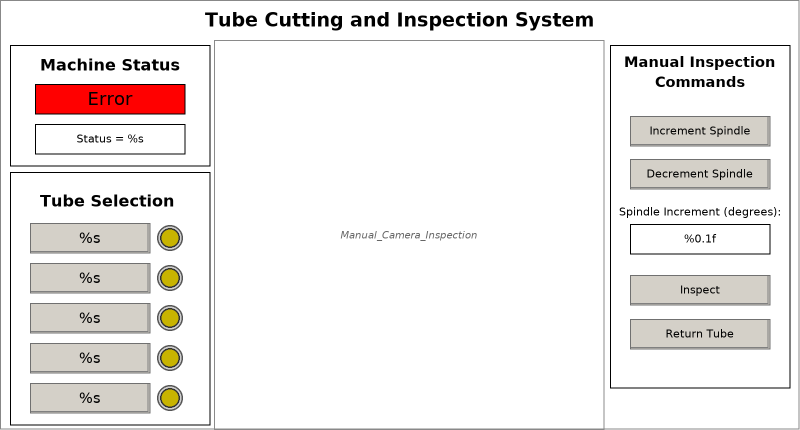
VISUALIZATION Manual_Inspect  // 800x430
    Rectangle (610,45 180x343)
    Frame (214,40 390x390)
        shows Manual_Camera_Inspection()
    Rectangle (10,172 200x253)
    Label (10,186 200x30), "Tube Selection"
    Button (30,223 120x30), "%s", text variable: MAIN.TubeSelection[1].ProductName
        OnMouseClick: execute {
            MAIN.TubeIndicator[1] := TRUE;
            MAIN.TubeIndicator[2] := FALSE;
            MAIN.TubeIndicator[3] := FALSE;
            MAIN.TubeIndicator[4] := FALSE;
            MAIN.TubeIndicator[5] := FALSE;
        }
    Button (30,263 120x30), "%s", text variable: MAIN.TubeSelection[2].ProductName
        OnMouseClick: execute {
            MAIN.TubeIndicator[1] := FALSE;
            MAIN.TubeIndicator[2] := TRUE;
            MAIN.TubeIndicator[3] := FALSE;
            MAIN.TubeIndicator[4] := FALSE;
            MAIN.TubeIndicator[5] := FALSE;
        }
    Button (30,303 120x30), "%s", text variable: MAIN.TubeSelection[3].ProductName
        OnMouseClick: execute {
            MAIN.TubeIndicator[1] := FALSE;
            MAIN.TubeIndicator[2] := FALSE;
            MAIN.TubeIndicator[3] := TRUE;
            MAIN.TubeIndicator[4] := FALSE;
            MAIN.TubeIndicator[5] := FALSE;
        }
    Button (30,343 120x30), "%s", text variable: MAIN.TubeSelection[4].ProductName, input disabled if: TRUE
        OnMouseClick: execute {
            MAIN.TubeIndicator[1] := FALSE;
            MAIN.TubeIndicator[2] := FALSE;
            MAIN.TubeIndicator[3] := FALSE;
            MAIN.TubeIndicator[4] := TRUE;
            MAIN.TubeIndicator[5] := FALSE;
        }
    Button (30,383 120x30), "%s", text variable: MAIN.TubeSelection[5].ProductName, input disabled if: TRUE
        OnMouseClick: execute {
            MAIN.TubeIndicator[1] := FALSE;
            MAIN.TubeIndicator[2] := FALSE;
            MAIN.TubeIndicator[3] := FALSE;
            MAIN.TubeIndicator[4] := FALSE;
            MAIN.TubeIndicator[5] := TRUE;
        }
    Lamp1 (155,223 30x30), variable: MAIN.TubeIndicator[1], style: Lamp-Lamp1-Yellow
    Lamp1 (155,263 30x30), variable: MAIN.TubeIndicator[2], style: Lamp-Lamp1-Yellow
    Lamp1 (155,303 30x30), variable: MAIN.TubeIndicator[3], style: Lamp-Lamp1-Yellow
    Lamp1 (155,343 30x30), variable: MAIN.TubeIndicator[4], style: Lamp-Lamp1-Yellow
    Lamp1 (155,383 30x30), variable: MAIN.TubeIndicator[5], style: Lamp-Lamp1-Yellow
    Label (0,5 800x30), "Tube Cutting and Inspection System"
    Rectangle (10,45 200x121)
    Label (10,50 200x30), "Machine Status"
    Rectangle (35,84 150x30), "Initializing", invisible if: MAIN.eState <> E_PMLState.ePMLState_Clearing
    Rectangle (35,84 150x30), "Ready", invisible if: MAIN.eState <> E_PMLState.ePMLState_Idle
    Rectangle (35,84 150x30), "Running", invisible if: MAIN.eState <> E_PMLState.ePMLState_Execute
    Rectangle (35,84 150x30), "Error", invisible if: MAIN.eState <> E_PMLState.ePMLState_Aborted
    Rectangle (35,124 150x30), "Status = %s", text variable: MAIN.hmiStatus
    Button (630,116 140x30), "Increment Spindle"
        tap MAIN.InspectCommands.IncrementSpindle
        OnMouseClick: execute { MAIN.fbSlitter.bIncrementSpindle := TRUE; }
    Button (630,275 140x30), "Inspect"
        tap MAIN.InspectCommands.Inspect
        OnMouseClick: execute { MAIN.fbSlitter.bInspect := TRUE; }
    Label (610,47 180x30), "Manual Inspection"
    Label (610,67 180x30), "Commands"
    Button (630,159 140x30), "Decrement Spindle"
        tap MAIN.InspectCommands.DecrementSpindle
        OnMouseClick: execute { MAIN.fbSlitter.bDecrementSpindle := TRUE; }
    Button (630,319 140x30), "Return Tube"
        tap MAIN.InspectCommands.InspectComplete
        OnMouseClick: execute { MAIN.fbSlitter.bInspectComplete := TRUE; }
    Rectangle (630,224 140x30), "%0.1f", text variable: MAIN.fbSlitter.Mandrel._SpindleIncrement
        OnMouseClick: write MAIN.fbSlitter.Mandrel._SpindleIncrement via Default
    Label (620,197 160x30), "Spindle Increment (degrees):"
END_VISUALIZATION

(* stored: Version 1.1.0.1, ProductVersion 3.1.4024.3
   Visu Manual_Inspect: Id {2784a428-5965-49a3-814f-ce0b6e8a6ebf} *)
